ABB RAPID module: A067_DataTask_Rob.mod

MODULE A067_DataTask_Rob
    !***********************************************************************************
    !
    ! ETH Zurich / NCCR Digital Fabrication
    ! HIB C51 / Stefano-Franscini-Platz 1
    ! CH-8093 Zurich
    !
    !***********************************************************************************
    !
    ! PROJECT     :  A067 Integral Timber Joints
    !
    ! FUNCTION    :  Includ all Task Data's for Project
    !
    ! AUTHOR      :  Philippe Fleischmann
    !
    ! EMAIL       :  fleischmann@arch.ethz.ch
    !
    ! HISTORY     :  2019.12.04
    !
    ! Copyright   :  ETH Zurich (CH) 2019
    !
    !***********************************************************************************

    !************************************************
    ! Declaration :     bool
    !************************************************
    !

    !************************************************
    ! Declaration :     num
    !************************************************
    !

    !************************************************
    ! Declaration :     string
    !************************************************
    !

    !************************************************
    ! Declaration :     tooldata
    !************************************************
    !
    TASK PERS tooldata t_A067_Tool:=[TRUE,[[0,0,0],[1,0,0,0]],[0,[0,0,0],[1,0,0,0],0,0,0]];
    TASK PERS tooldata t_A067_T1_Gripper:=[TRUE,[[0,0,0],[1,0,0,0]],[10,[0,0,150],[1,0,0,0],0,0,0]];

    !************************************************
    ! Declaration :     wobjdata
    !************************************************
    !
    TASK PERS wobjdata ob_A067_Wobjdata:=[FALSE,TRUE,"",[[0,0,0],[1,0,0,0]],[[0,0,0],[1,0,0,0]]];

    !************************************************
    ! Declaration :     robtarget
    !************************************************
    !
    TASK PERS robtarget p_A067_Robtarget:=[[0,0,0],[1,0,0,0],[0,0,0,0],[9E9,9E9,9E9,9E9,9E9,9E9]];

    !************************************************
    ! Declaration :     speeddata
    !************************************************
    !
    TASK PERS speeddata v_A067_Speed:=[0,0,0,0];

ENDMODULE
